FUNCTION_BLOCK FB_HE_SATT_UserRequest_Test EXTENDS FB_TestSuite
VAR
END_VAR


GivenApplyCommandedStartNewConfiguration();


METHOD PRIVATE GivenApplyCommandedStartNewConfiguration
VAR
    fbHE_SATT_SequenceTestDouble : FB_HE_SATT_SequenceTestDouble;
    
    // Subject under test
    fbHE_SATT_UserRequest : FB_HE_SATT_UserRequest(iHE_SATT_Sequence := fbHE_SATT_SequenceTestDouble);
END_VAR

TEST('GivenApplyCommandedStartNewConfiguration');

fbHE_SATT_UserRequest.RequestTransmission(
    fRequestedTransmission := 0.8,
    eRequestedRoundingMode := E_HE_SATT_RoundingMode.CEIL_WITHIN_TOLERANCE,
    fRequestedAllowableTolerance := 1e-2
);

AssertEquals_LREAL(
    Expected := 0.0,
    Actual := fbHE_SATT_SequenceTestDouble.GetStartTransmissionValue(),
    Delta := 0.0001,
    Message := 'Not correct value #1'
);

AssertEquals_UINT(
    Expected := E_HE_SATT_RoundingMode.FLOOR_WITHIN_TOLERANCE,
    Actual := fbHE_SATT_SequenceTestDouble.GetStartRoundingModeValue(),
    Message := 'Not correct value #2'
);

AssertEquals_LREAL(
    Expected := 0.0,
    Actual := fbHE_SATT_SequenceTestDouble.GetStartAllowableToleranceValue(),
    Delta := 0.0001,
    Message := 'Not correct value #3'
);

fbHE_SATT_UserRequest.ApplyConfig();

AssertEquals_LREAL(
    Expected := 0.8,
    Actual := fbHE_SATT_SequenceTestDouble.GetStartTransmissionValue(),
    Delta := 0.0001,
    Message := 'Not correct value #4'
);

AssertEquals_UINT(
    Expected := E_HE_SATT_RoundingMode.CEIL_WITHIN_TOLERANCE,
    Actual := fbHE_SATT_SequenceTestDouble.GetStartRoundingModeValue(),
    Message := 'Not correct value #5'
);

AssertEquals_LREAL(
    Expected := 1e-2,
    Actual := fbHE_SATT_SequenceTestDouble.GetStartAllowableToleranceValue(),
    Delta := 0.0001,
    Message := 'Not correct value #6'
);

TEST_FINISHED();
END_METHOD

END_FUNCTION_BLOCK

(* stored: Version 1.1.0.1
   POU FB_HE_SATT_UserRequest_Test: Id {f725bdf0-5866-43db-ae0d-351577d2575d}, SpecialFunc None
   Method GivenApplyCommandedStartNewConfiguration: Id {066ac0f4-63b3-4282-91e3-be7ba1a2dd59} *)
